(*
Retrieves the I_Entity instance at the given nIndex from the global entity list.
Returns:
- Ok - Returns I_Entity
- None - Returns Null
*)
FUNCTION GetEntity : Result
VAR_INPUT
	nIndex		: UDINT;
END_VAR
VAR_OUTPUT
	iEntity		: I_Entity;
END_VAR

IF nIndex > _Ec.nEntityLen OR nIndex = 0 THEN
	GetEntity := None;
	RETURN;
END_IF

iEntity := _Ec.iEntity[nIndex]._AsIEntity;
GetEntity := Ok;

END_FUNCTION

(* stored: Version 1.1.0.1
   POU GetEntity: Id {f364a793-1b08-4c02-b87e-c6952bc10b65}, SpecialFunc None *)
